{attribute 'qualified_only'}
VAR_GLOBAL CONSTANT
    const115_01Y : AxisLinMotConst_t := (POS_MIN := -5, POS_MAX := 650, VELO_MAX := 2000, VELO_MANU := 100);
    const115_02Z : AxisLinMotConst_t := (POS_MIN := -5, POS_MAX := 650, VELO_MAX := 2000, VELO_MANU := 50);
    const115_03Z : AxisLinMotConst_t := (POS_MIN := -5, POS_MAX := 650, VELO_MAX := 2000, VELO_MANU := 50);
    const115_04Z : AxisLinMotConst_t := (POS_MIN := -5, POS_MAX := 650, VELO_MAX := 2000, VELO_MANU := 50);
    const115_10W : AxisLinMotConst_t := (POS_MIN := 0, POS_MAX := 360, VELO_MAX := 360, VELO_MANU := 50);

END_VAR
VAR_GLOBAL
    axis115_01Y : AxisLinMot_t;
    axis115_02Z : AxisBeckhoff_t;
    axis115_03Z : AxisBeckhoff_t;
    axis115_04Z : AxisBeckhoff_t;
    axis115_10W : AxisLinMot_t;
END_VAR
VAR_GLOBAL RETAIN
    // Recipe values are managed elsewhere
END_VAR

(* stored: Version 1.1.0.1, ProductVersion 3.1.4024.6
   GVL ST115_Axis: Id {f974398c-0773-40d2-bb5c-7d1fe23b7e79} *)
